// Mitsubishi GX Works2 project: final - Copy   PLC: FX3G

// global labels: Global1
VAR_GLOBAL
  system_1_start AT X010 : BOOL;
  system_1_stop AT X005 : BOOL;
  sen_pallet AT X001 : BOOL;
  sen_30 AT X002 : BOOL;
  sen_15 AT X003 : BOOL;
  sen_spray AT X004 : BOOL;
END_VAR
VAR_GLOBAL CONSTANT
  cookie : INT := 6;
  cream : INT := 300;
  chocolate : INT := 120;
END_VAR
VAR_GLOBAL
  spray AT Y004 : BOOL;
  system_1_on AT M0 : BOOL;
  spray_to_chocolate1 AT Y000 : BOOL;
  spray_to_chocolate2 AT Y001 : BOOL;
  flash_light1 AT TS1 : BOOL;
  flash_light2 AT TS2 : BOOL;
  tc_1 AT TC1 : BOOL;
  tc_2 AT TC2 : BOOL;
END_VAR
VAR_GLOBAL CONSTANT
  K_light : INT := 5;
END_VAR
VAR_GLOBAL
  M_2 AT M2 : BOOL;
  M_3 AT M3 : BOOL;
  TC_3 AT TC3 : BOOL;
  TS_3 AT TS3 : BOOL;
END_VAR
VAR_GLOBAL CONSTANT
  K_flash : INT := 40;
END_VAR
VAR_GLOBAL
  flashing AT M1 : BOOL;
  day_light AT Y007 : BOOL;
  cookie_stash AT D1100 : INT;
  cream_stash AT D1110 : INT;
  chocolate_stash AT D1120 : INT;
  start_day AT X007 : BOOL;
  stage1_start AT X011 : BOOL;
  cookie_count AT CC1 : BOOL;
  cream_count AT CC2 : BOOL;
  chocolate_count AT CC3 : BOOL;
  cookie_count_resault AT CS1 : BOOL;
  cream_count_resault AT CS2 : BOOL;
  chocolate_count_resault AT CS3 : BOOL;
  start_glazing_process AT X006 : BOOL;
  end_day AT M6 : BOOL;
  TC_4 AT TC4 : BOOL;
  TS_4 AT TS4 : BOOL;
  TC_5 AT TC5 : BOOL;
  TS_5 AT TS5 : BOOL;
  TC_6 AT TC6 : BOOL;
  TS_6 AT TS6 : BOOL;
  M_10 AT M10 : BOOL;
  M_11 AT M11 : BOOL;
  M_12 AT M12 : BOOL;
END_VAR
VAR_GLOBAL CONSTANT
  regular_glazing_upper_limit : INT := 2000;
  double_glazing_lower_limit : INT := 2400;
  double_glazing_upper_limit : INT := 4000;
  wrapped_all_Crembos : INT := 6;
  wrapped_5_Crembos : INT := 5;
  Cremos_in_pack : REAL := 6;
  diiv_Crembos : INT := 10;
END_VAR
VAR_GLOBAL
  M_13 AT M13 : BOOL;
  M_14 AT M14 : BOOL;
  M_15 AT M15 : BOOL;
END_VAR
VAR_GLOBAL CONSTANT
  end_day_flashi : INT := 30;
END_VAR
VAR_GLOBAL
  Analog_input1 AT D8280 : INT;
  glazing_timer AT TC10 : BOOL;
  glazing_TS AT TS10 : BOOL;
  Crembo_counter_for_5 AT CC10 : BOOL;
  fifth_Crembo AT CS10 : BOOL;
  sixth_Crembo AT CS13 : BOOL;
  Crembos_counter_for_6 AT CC13 : BOOL;
  Analog_output AT D8282 : INT;
  totalCrembos AT D1200 : REAL;
  we_are_glazing AT Y003 : BOOL;
  wrap_1_Crembo AT X000 : BOOL;
  wrapped_5_light AT Y002 : BOOL;
  regular_glaze AT M16 : BOOL;
  double_glaze_1 AT M17 : BOOL;
  start_coating AT M18 : BOOL;
  send_to_wrap AT M19 : BOOL;
  end_of_the_day AT M20 : BOOL;
END_VAR
VAR_GLOBAL CONSTANT
  double_topping : INT := 2;
  regular_topping : INT := 1;
  divCrembos : INT := 10;
  glazing_time : INT := 50;
END_VAR
VAR_GLOBAL
  finish_wrap AT M21 : BOOL;
END_VAR
VAR_GLOBAL CONSTANT
  for_output : REAL := 40.0;
END_VAR
VAR_GLOBAL
  output_mul AT D1400 : REAL;
  chocolate_can_start AT M22 : BOOL;
  glazing_done AT M23 : BOOL;
  stash_light AT M27 : BOOL;
  temp_output AT M25 : BOOL;
  system1_ready AT M26 : BOOL;
  double_glaze_2 AT M24 : BOOL;
  input_cream AT D1130 : INT;
  input_cookie AT D1140 : INT;
  input_chocolate AT D1150 : INT;
  dip_chocolate AT D1600 : INT;
  pour_cream AT D1610 : INT;
  cookie_amount AT D1300 : INT;
  chocolate_amount AT D1310 : INT;
  cream_amount AT D1320 : INT;
END_VAR
VAR_GLOBAL CONSTANT
  double_chocolate : INT := 240;
  zero : INT;
END_VAR
VAR_GLOBAL
  no_chocolate AT M30 : BOOL;
END_VAR

// task Task_01 (event TRUE, interval 0, priority 31): POU_01

PROGRAM POU_01
(* structured ladder/FBD written out as ST: instructions are called as NAME(EN, inputs, outputs); _pN, _eN, _tN stand for wires *)
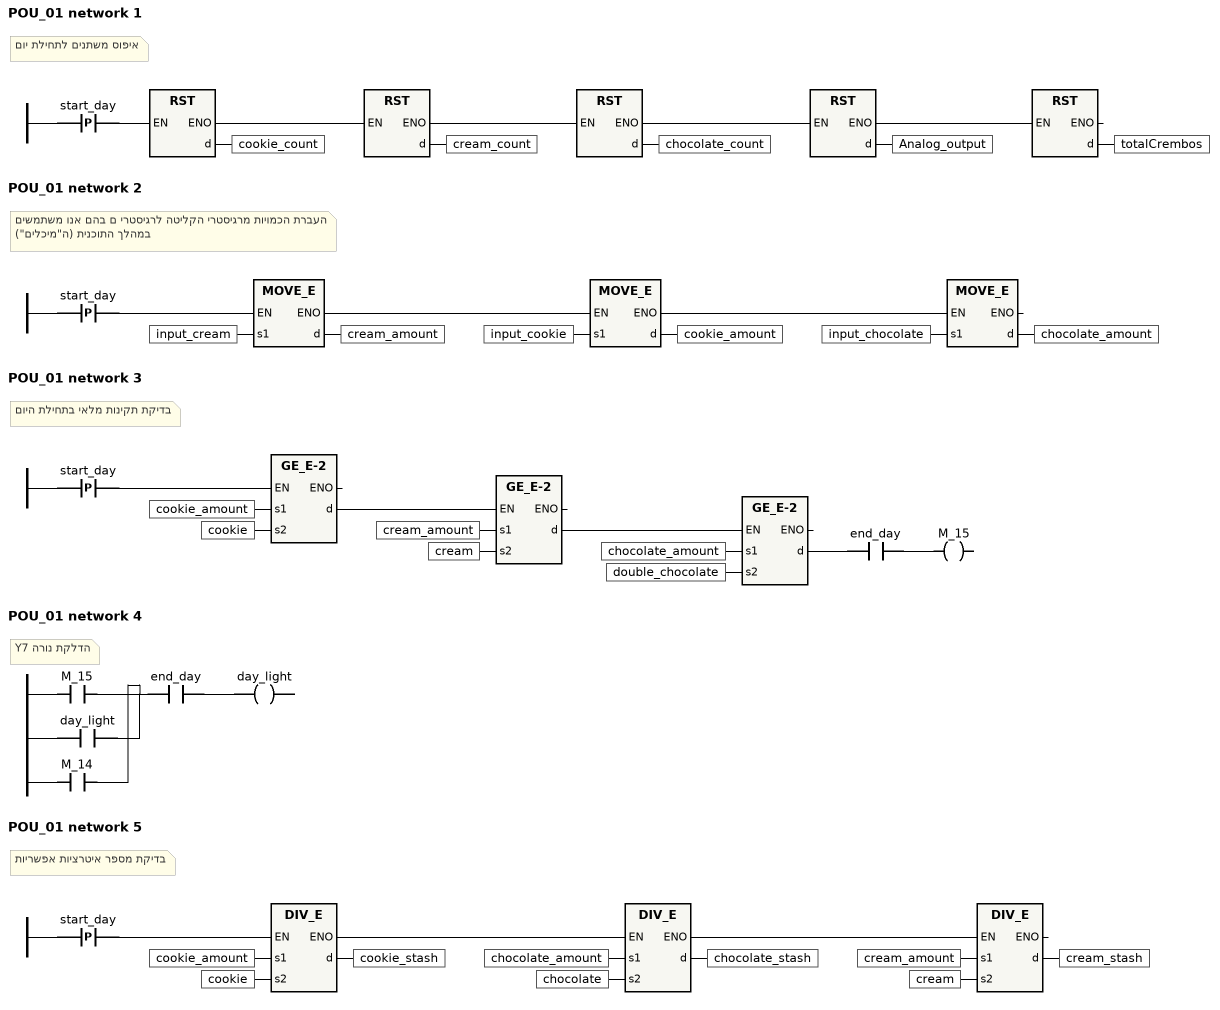
(* network 1 *)
(* איפוס משתנים לתחילת יום *)
_e1 := RST(LDP(TRUE, start_day), cookie_count);
_e2 := RST(_e1, cream_count);
_e3 := RST(_e2, chocolate_count);
_e4 := RST(_e3, Analog_output);
RST(_e4, totalCrembos);
(* network 2 *)
(* העברת הכמויות מרגיסטרי הקליטה לרגיסטרי ם בהם אנו משתמשים במהלך התוכנית (ה"מיכלים") *)
_e1 := MOVE_E(LDP(TRUE, start_day), input_cream, cream_amount);
_e2 := MOVE_E(_e1, input_cookie, cookie_amount);
MOVE_E(_e2, input_chocolate, chocolate_amount);
(* network 3 *)
(* בדיקת תקינות מלאי בתחילת היום *)
GE_E(LDP(TRUE, start_day), cookie_amount, cookie, _t1);
GE_E(_t1, cream_amount, cream, _t2);
GE_E(_t2, chocolate_amount, double_chocolate, _t3);
M_15 := _t3 AND end_day;
(* network 4 *)
(* הדלקת נורה Y7 *)
day_light := (M_15 OR day_light OR M_14) AND end_day;
(* network 5 *)
(* בדיקת מספר איטרציות אפשריות *)
_e1 := DIV_E(LDP(TRUE, start_day), cookie_amount, cookie, cookie_stash);
_e2 := DIV_E(_e1, chocolate_amount, chocolate, chocolate_stash);
DIV_E(_e2, cream_amount, cream, cream_stash);
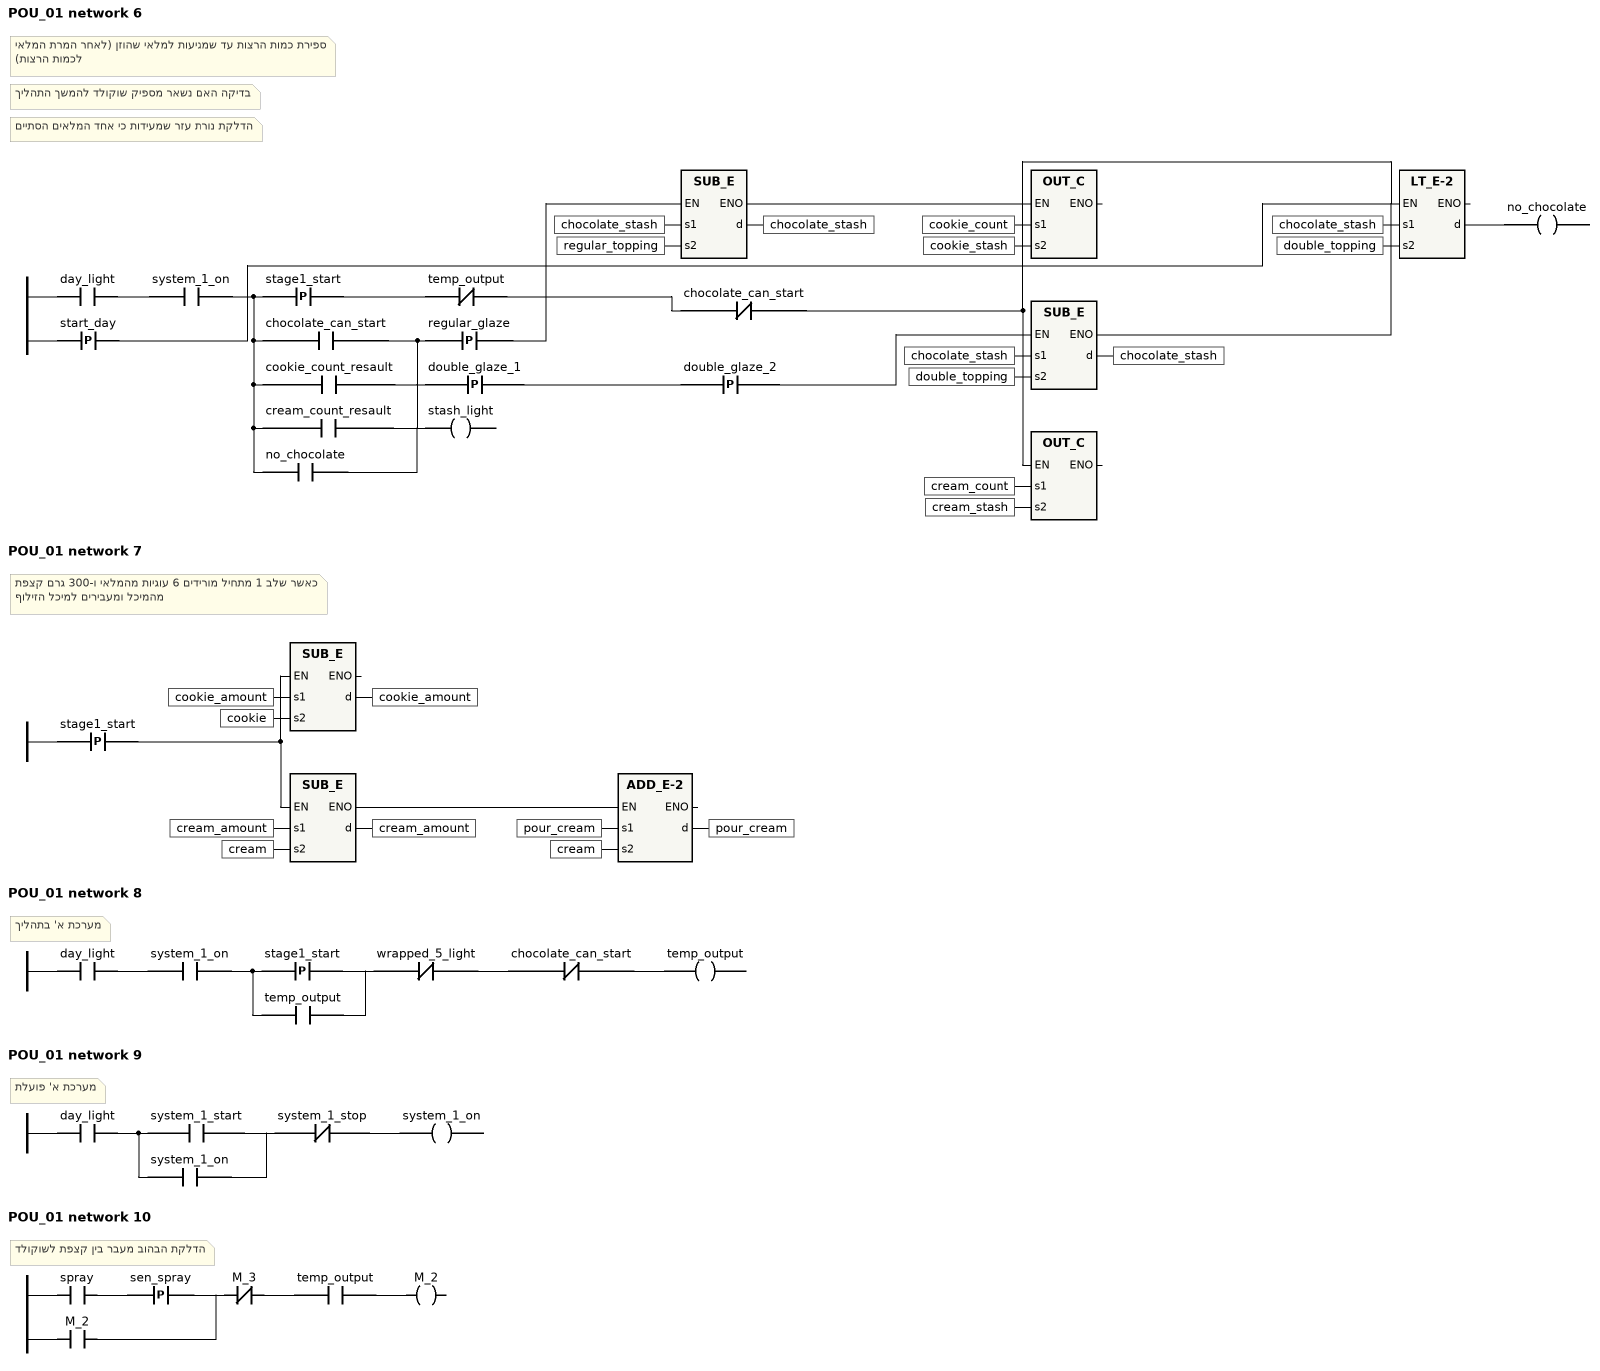
(* network 6 *)
(* ספירת כמות הרצות עד שמגיעות למלאי שהוזן (לאחר המרת המלאי לכמות הרצות) *)
(* בדיקה האם נשאר מספיק שוקולד להמשך התהליך *)
(* הדלקת נורת עזר שמעידות כי אחד המלאים הסתיים *)
_p1 := day_light AND system_1_on;
_p2 := _p1 AND LDP(TRUE, stage1_start) AND NOT temp_output AND NOT chocolate_can_start;
OUT_C(_p2, cookie_count, cookie_stash);
OUT_C(_p2, cream_count, cream_stash);
_p3 := _p1 AND chocolate_can_start;
_e4 := SUB_E(_p3 AND LDP(TRUE, regular_glaze), chocolate_stash, regular_topping, chocolate_stash);
_e5 := SUB_E(_p3 AND LDP(TRUE, double_glaze_1) AND LDP(TRUE, double_glaze_2), chocolate_stash, double_topping, chocolate_stash);
LT_E(LDP(TRUE, start_day) OR _e4 OR _e5, chocolate_stash, double_topping, _t6);
no_chocolate := _t6;
stash_light := (_p1 AND cookie_count_resault) OR (_p1 AND cream_count_resault) OR (_p1 AND no_chocolate);
(* network 7 *)
(* כאשר שלב 1 מתחיל מורידים 6 עוגיות מהמלאי ו-300 גרם קצפת מהמיכל ומעבירים למיכל הזילוף *)
_p1 := LDP(TRUE, stage1_start);
SUB_E(_p1, cookie_amount, cookie, cookie_amount);
_e2 := SUB_E(_p1, cream_amount, cream, cream_amount);
ADD_E(_e2, pour_cream, cream, pour_cream);
(* network 8 *)
(* מערכת א' בתהליך *)
_p1 := day_light AND system_1_on;
temp_output := (((_p1 AND LDP(TRUE, stage1_start)) OR (_p1 AND temp_output)) AND NOT wrapped_5_light) AND NOT chocolate_can_start;
(* network 9 *)
(* מערכת א' פועלת *)
system_1_on := ((day_light AND system_1_start) OR (day_light AND system_1_on)) AND NOT system_1_stop;
(* network 10 *)
(* הדלקת הבהוב מעבר בין קצפת לשוקולד *)
M_2 := (((spray AND LDP(TRUE, sen_spray)) OR M_2) AND NOT M_3) AND temp_output;
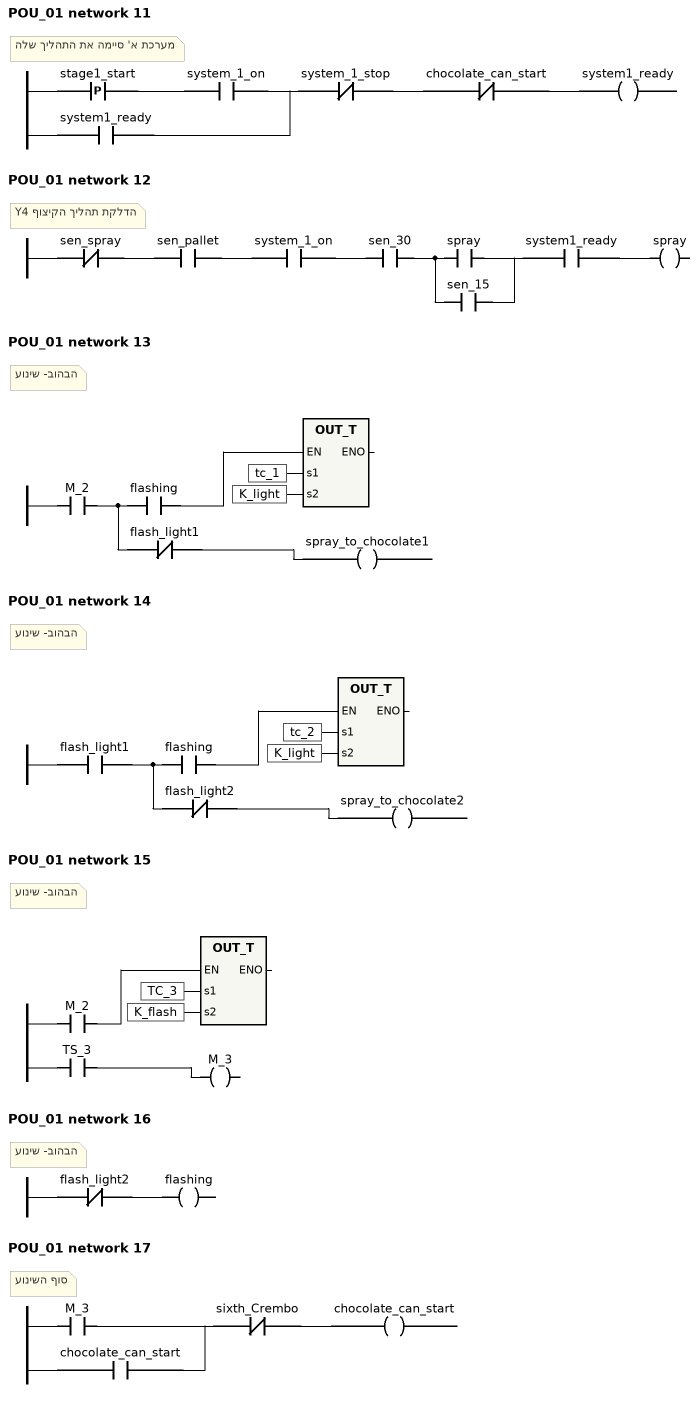
(* network 11 *)
(* מערכת א' סיימה את התהליך שלה *)
system1_ready := (((LDP(TRUE, stage1_start) AND system_1_on) OR system1_ready) AND NOT system_1_stop) AND NOT chocolate_can_start;
(* network 12 *)
(* Y4 הדלקת תהליך הקיצוף *)
_p1 := NOT sen_spray AND sen_pallet AND system_1_on AND sen_30;
spray := ((_p1 AND spray) OR (_p1 AND sen_15)) AND system1_ready;
(* network 13 *)
(* הבהוב- שינוע *)
OUT_T(M_2 AND flashing, tc_1, K_light);
spray_to_chocolate1 := M_2 AND NOT flash_light1;
(* network 14 *)
(* הבהוב- שינוע *)
OUT_T(flash_light1 AND flashing, tc_2, K_light);
spray_to_chocolate2 := flash_light1 AND NOT flash_light2;
(* network 15 *)
(* הבהוב- שינוע *)
OUT_T(M_2, TC_3, K_flash);
M_3 := TS_3;
(* network 16 *)
(* הבהוב- שינוע *)
flashing := NOT flash_light2;
(* network 17 *)
(* סוף השינוע *)
chocolate_can_start := (M_3 OR chocolate_can_start) AND NOT sixth_Crembo;
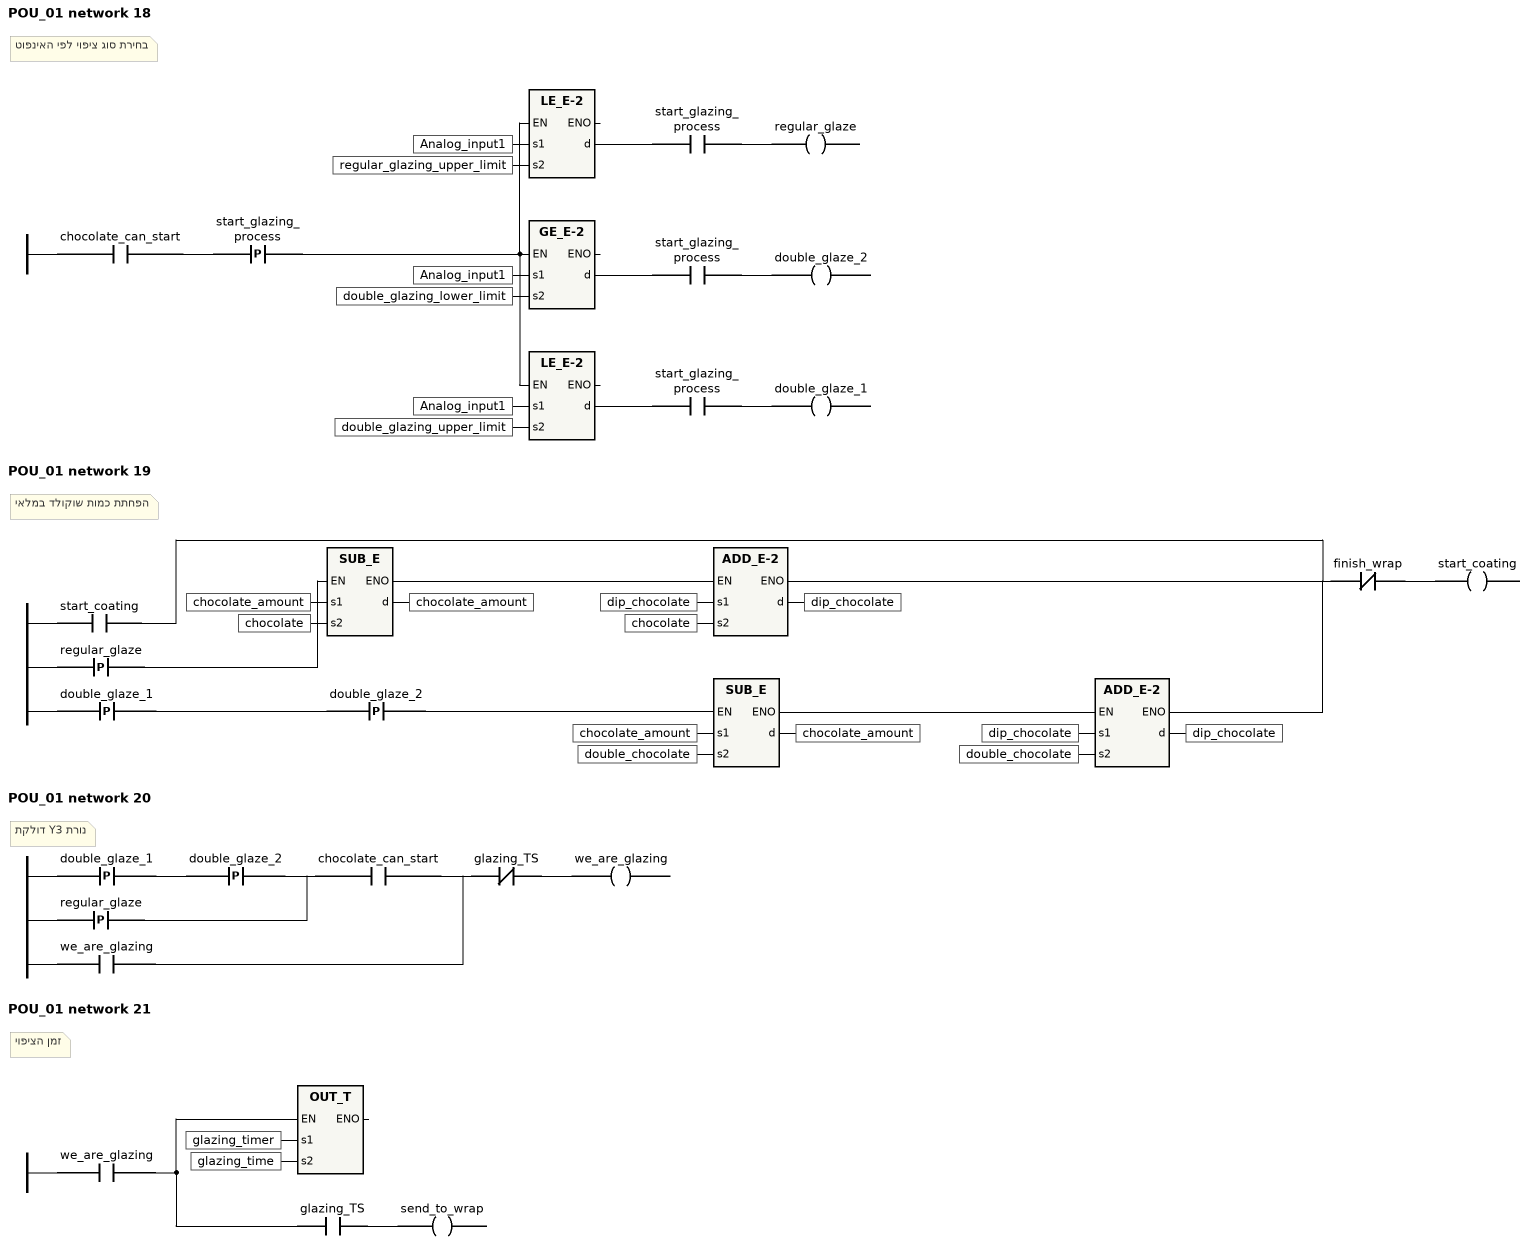
(* network 18 *)
(* בחירת סוג ציפוי לפי האינפוט *)
_p1 := chocolate_can_start AND LDP(TRUE, start_glazing_process);
LE_E(_p1, Analog_input1, regular_glazing_upper_limit, _t2);
regular_glaze := _t2 AND start_glazing_process;
GE_E(_p1, Analog_input1, double_glazing_lower_limit, _t3);
double_glaze_2 := _t3 AND start_glazing_process;
LE_E(_p1, Analog_input1, double_glazing_upper_limit, _t4);
double_glaze_1 := _t4 AND start_glazing_process;
(* network 19 *)
(* הפחתת כמות שוקולד במלאי *)
_e1 := SUB_E(LDP(TRUE, regular_glaze), chocolate_amount, chocolate, chocolate_amount);
_e2 := ADD_E(_e1, dip_chocolate, chocolate, dip_chocolate);
_e3 := SUB_E(LDP(TRUE, double_glaze_1) AND LDP(TRUE, double_glaze_2), chocolate_amount, double_chocolate, chocolate_amount);
_e4 := ADD_E(_e3, dip_chocolate, double_chocolate, dip_chocolate);
start_coating := (start_coating OR _e2 OR _e4) AND NOT finish_wrap;
(* network 20 *)
(* נורת Y3 דולקת *)
we_are_glazing := ((((LDP(TRUE, double_glaze_1) AND LDP(TRUE, double_glaze_2)) OR LDP(TRUE, regular_glaze)) AND chocolate_can_start) OR we_are_glazing) AND NOT glazing_TS;
(* network 21 *)
(* זמן הציפוי *)
OUT_T(we_are_glazing, glazing_timer, glazing_time);
send_to_wrap := we_are_glazing AND glazing_TS;
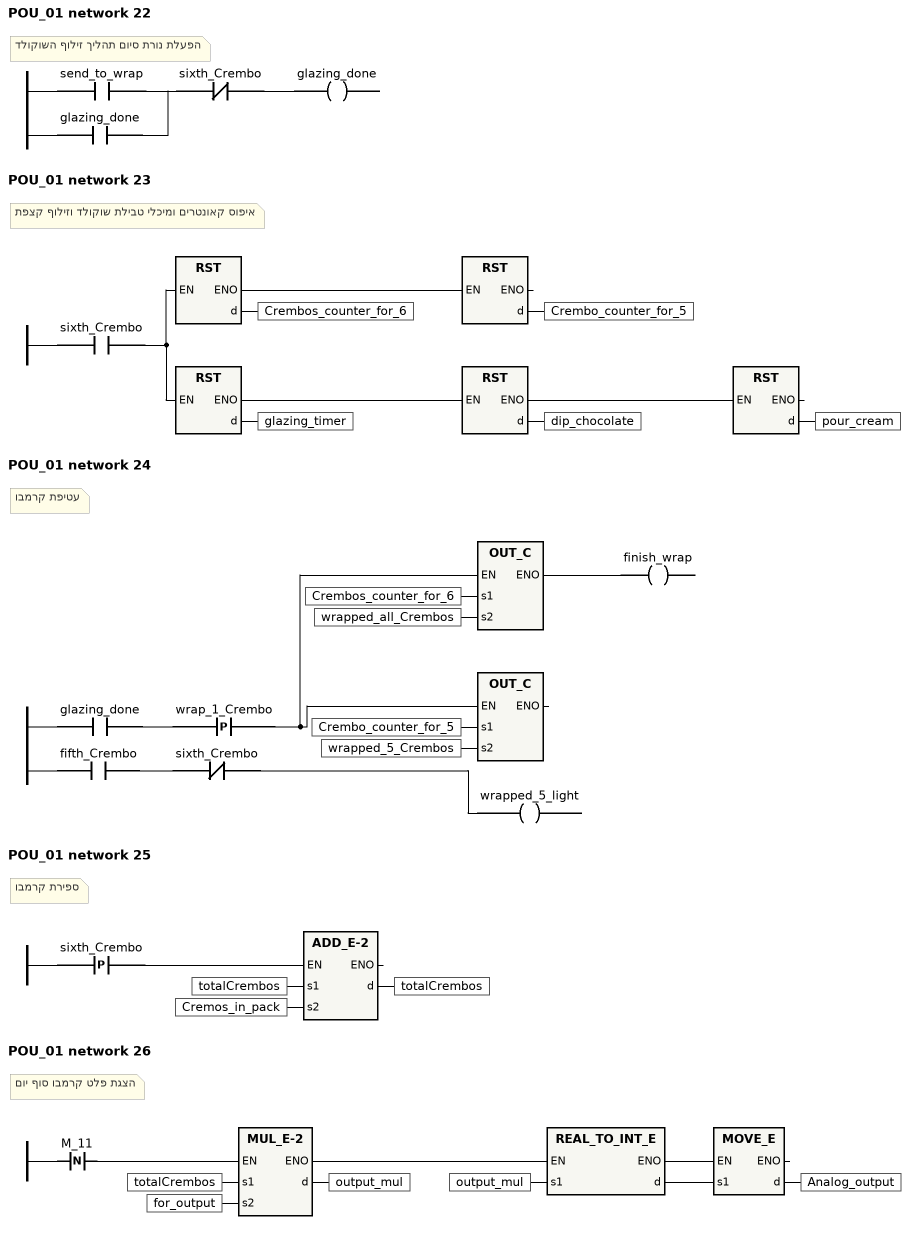
(* network 22 *)
(* הפעלת נורת סיום תהליך זילוף השוקולד *)
glazing_done := (send_to_wrap OR glazing_done) AND NOT sixth_Crembo;
(* network 23 *)
(* איפוס קאונטרים ומיכלי טבילת שוקולד וזילוף קצפת *)
_e1 := RST(sixth_Crembo, Crembos_counter_for_6);
RST(_e1, Crembo_counter_for_5);
_e2 := RST(sixth_Crembo, glazing_timer);
_e3 := RST(_e2, dip_chocolate);
RST(_e3, pour_cream);
(* network 24 *)
(* עטיפת קרמבו *)
_p1 := glazing_done AND LDP(TRUE, wrap_1_Crembo);
OUT_C(_p1, Crembo_counter_for_5, wrapped_5_Crembos);
_e2 := OUT_C(_p1, Crembos_counter_for_6, wrapped_all_Crembos);
finish_wrap := _e2;
wrapped_5_light := fifth_Crembo AND NOT sixth_Crembo;
(* network 25 *)
(* ספירת קרמבו *)
ADD_E(LDP(TRUE, sixth_Crembo), totalCrembos, Cremos_in_pack, totalCrembos);
(* network 26 *)
(* הצגת פלט קרמבו סוף יום *)
_e1 := MUL_E(LDF(TRUE, M_11), totalCrembos, for_output, output_mul);
_e3 := REAL_TO_INT_E(_e1, output_mul, _t2);
MOVE_E(_e3, _t2, Analog_output);
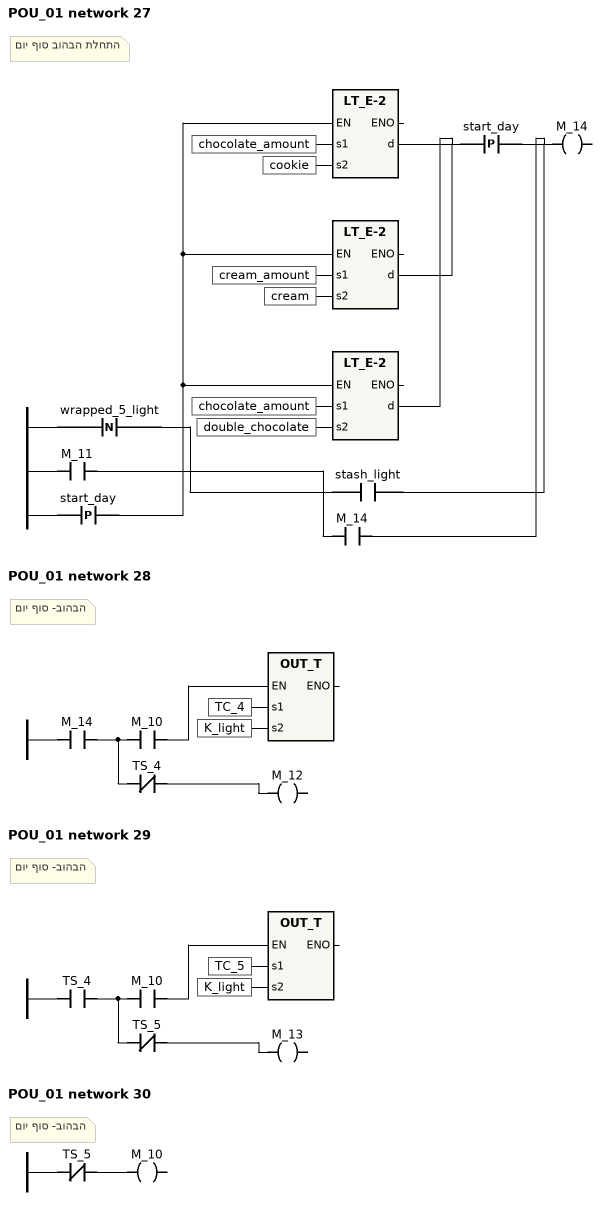
(* network 27 *)
(* התחלת הבהוב סוף יום *)
_p1 := LDP(TRUE, start_day);
LT_E(_p1, chocolate_amount, cookie, _t2);
LT_E(_p1, cream_amount, cream, _t3);
LT_E(_p1, chocolate_amount, double_chocolate, _t4);
M_14 := (LDF(TRUE, wrapped_5_light) AND stash_light) OR (M_11 AND M_14) OR ((_t2 OR _t3 OR _t4) AND LDP(TRUE, start_day));
(* network 28 *)
(* הבהוב- סוף יום *)
OUT_T(M_14 AND M_10, TC_4, K_light);
M_12 := M_14 AND NOT TS_4;
(* network 29 *)
(* הבהוב- סוף יום *)
OUT_T(TS_4 AND M_10, TC_5, K_light);
M_13 := TS_4 AND NOT TS_5;
(* network 30 *)
(* הבהוב- סוף יום *)
M_10 := NOT TS_5;
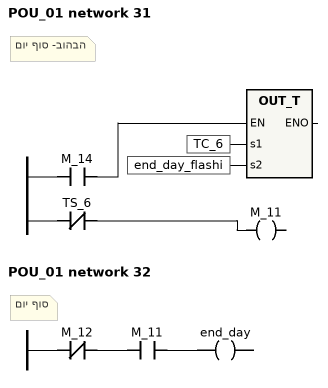
(* network 31 *)
(* הבהוב- סוף יום *)
OUT_T(M_14, TC_6, end_day_flashi);
M_11 := NOT TS_6;
(* network 32 *)
(* סוף יום *)
end_day := NOT M_12 AND M_11;
END_PROGRAM
